{attribute addProperty BoxType "EK1122-0000-0018"}
{attribute addProperty Id "Beckhoff_EQ2xxxsub_EK1100EK1100_179A0949162A_0001_EQ2008_0002_0016EQ2008_A854BE6D8110.125A_0002_EQ2008_0002_0017EQ2008_A854BE6D8110.125A_0003_EQ2008_0002_0018EQ2008_A854BE6D8110.125A_0004_EQ2008_0002_0019EQ2008_A854BE6D8110.125A_0005_EQ2339_0022_0016EQ2339_9219B49827434.25A_0006_EQ2339_0022_0017EQ2339_9219B49827434.25A_0007_EQ2339_0022_0018EQ2339_9219B49827434.25A_0008_EQ2339_0022_0019EQ2339_9219B49827434.25A_0009_EQ2809_0022_0016EQ2809_859F43D214518.125A_0010_EQ2809_0022_0017EQ2809_859F43D214518.125A_0011_EQ2809_0022_0018EQ2809_859F43D214518.125"}
{attribute addProperty CRC "1621022759"}
{attribute addProperty SizeInBites "1871"}
{attribute addProperty SizeInBytes "233.875"}
TYPE Beckhoff_EQ2xxxEK1122_609ED827 EXTENDS EK1122_179A0949 :
STRUCT
	{attribute addProperty Name "Beckhoff_EQ2xxxsub_EK1100"}
	Beckhoff_EQ2xxxsub_EK1100 : EK1100_179A0949;
	{attribute addProperty Name "A_0001_EQ2008_0002_0016"}
	A_0001_EQ2008_0002_0016 : EQ2008_A854BE6D;
	{attribute addProperty Name "A_0002_EQ2008_0002_0017"}
	A_0002_EQ2008_0002_0017 : EQ2008_A854BE6D;
	{attribute addProperty Name "A_0003_EQ2008_0002_0018"}
	A_0003_EQ2008_0002_0018 : EQ2008_A854BE6D;
	{attribute addProperty Name "A_0004_EQ2008_0002_0019"}
	A_0004_EQ2008_0002_0019 : EQ2008_A854BE6D;
	{attribute addProperty Name "A_0005_EQ2339_0022_0016"}
	A_0005_EQ2339_0022_0016 : EQ2339_9219B498;
	{attribute addProperty Name "A_0006_EQ2339_0022_0017"}
	A_0006_EQ2339_0022_0017 : EQ2339_9219B498;
	{attribute addProperty Name "A_0007_EQ2339_0022_0018"}
	A_0007_EQ2339_0022_0018 : EQ2339_9219B498;
	{attribute addProperty Name "A_0008_EQ2339_0022_0019"}
	A_0008_EQ2339_0022_0019 : EQ2339_9219B498;
	{attribute addProperty Name "A_0009_EQ2809_0022_0016"}
	A_0009_EQ2809_0022_0016 : EQ2809_859F43D2;
	{attribute addProperty Name "A_0010_EQ2809_0022_0017"}
	A_0010_EQ2809_0022_0017 : EQ2809_859F43D2;
	{attribute addProperty Name "A_0011_EQ2809_0022_0018"}
	A_0011_EQ2809_0022_0018 : EQ2809_859F43D2;
END_STRUCT
END_TYPE

(* stored: Version 1.2.0.0, ProductVersion 3.1.4024.9
   DUT Beckhoff_EQ2xxxEK1122_609ED827: Id {74e2e49e-4eed-46fe-b7a0-ede8fd0dcfc5} *)
